TYPE (* ButtonActivationCode Struct *)
  (* Version 1.0, 2025-07-21, Franz Höpfinger, initial API and implementation and/or initial documentation *)
  PACKAGE isobus::UT::io::Button;
  IMPORT eclipse4diac::core::TypeHash;
  ButtonActivationCode_S : STRUCT
    code : USINT := 255;
    bCyclic : BOOL := TRUE; (* do not repeat every 200ms if this is set FALSE *)
  END_STRUCT;
END_TYPE
